(* CODESYS project stepworker_1044.library
   Author: Boido
   Placeholder: StepWorkerLib
   Title: StepWorkerLib
   Version: 1.0.4.4
   Company: FactoryAutomation

Project tree, tasks and I/O mapping:
  libraries: Tc2_Standard, * (Beckhoff Automation GmbH); Tc2_System, * (Beckhoff Automation GmbH); Tc2_Utilities, * (Beckhoff Automation GmbH); Tc3_Module, * (Beckhoff Automation GmbH); VersionLib, * (FactoryAutomation)
  DUTs/
  GVLs/
  POUs/
    function block Actuator [ST]
    function block Boolean [ST]: getValue, setValue
    function block BoolIn [ST]: CallAfterInit, getValue, setValue
    function block BoolOut [ST]: CallAfterInit, getValue, setValue
    function block FB_StepWorker [ST]: getStep, mAddCondition, mConfigureTimeout, mNextStep
    interface I_Comparator: mEquals, mGreaterEquals, mGreaterThan, mLessEquals, mLessThan
    interface I_StepCondition: getValue, setValue
    interface I_StepWorker: mAddCondition
    function block IntComparator [ST]: getValue, mEquals, mGreaterEquals, mGreaterThan, mLessEquals, mLessThan, setValue
    function block LrealComparator [ST]: getValue, mEquals, mGreaterEquals, mGreaterThan, mLessEquals, mLessThan, setValue
    program MAIN [ST]
    function block RealComparator [ST]: getValue, mEquals, mGreaterEquals, mGreaterThan, mLessEquals, mLessThan, setValue
    function block SymbolPathStorage [ST]
    function block UintComparator [ST]: getValue, mEquals, mGreaterEquals, mGreaterThan, mLessEquals, mLessThan, setValue
  VISUs/
  program Version [ST]
*)

// POUs/Actuator
FUNCTION_BLOCK Actuator
VAR_INPUT
END_VAR
VAR_OUTPUT
	fbOutput : BoolOut;
END_VAR
VAR
END_VAR

END_FUNCTION_BLOCK

// POUs/BoolOut
{attribute 'call_after_init'}
{attribute 'reflection'}
FUNCTION_BLOCK PUBLIC BoolOut EXTENDS SymbolPathStorage IMPLEMENTS I_StepCondition
VAR_INPUT
END_VAR
VAR_OUTPUT
END_VAR
VAR
	{attribute 'instance-path'}  
	{attribute 'no_init'} 
	sPath : STRING;
	bValue AT%Q* : BOOL;
	sInitPath : STRING;

END_VAR

{attribute 'call_after_init'}
METHOD PRIVATE CallAfterInit : BOOL
IF uiPathCounter <= cMaxPaths 
THEN
	//Delete the part of the path which contains solution and project name 	
	sInitPath := DELETE(sPath,FIND(sPath,'.'),1);
	sInitPath := DELETE(sInitPath,FIND(sInitPath,'.'),1);
	sInitPath := CONCAT(sInitPath,'.bValue');
	aPaths[uiPathCounter] := sInitPath;
	uiPathCounter := uiPathCounter + 1;
END_IF
END_METHOD


PROPERTY getValue : BOOL
GET
getValue := bValue;
END_GET
END_PROPERTY


PROPERTY setValue : BOOL
SET
bValue := setValue;
END_SET
END_PROPERTY

END_FUNCTION_BLOCK

// POUs/SymbolPathStorage
FUNCTION_BLOCK SymbolPathStorage

VAR_OUTPUT
END_VAR
VAR_STAT
	aPaths : ARRAY[1..cMaxPaths] OF STRING;
	uiPathCounter : UINT := 1;
END_VAR
VAR CONSTANT
	cMaxPaths : UINT := 512;
END_VAR

END_FUNCTION_BLOCK

// POUs/I_StepCondition
INTERFACE I_StepCondition

PROPERTY getValue : BOOL
GET
END_GET
END_PROPERTY

PROPERTY setValue : Bool
SET
END_SET
END_PROPERTY

END_INTERFACE

// POUs/Boolean
FUNCTION_BLOCK PUBLIC Boolean IMPLEMENTS I_StepCondition
VAR_INPUT
END_VAR
VAR_OUTPUT
END_VAR
VAR
	bValue : BOOL;
END_VAR

PROPERTY getValue : BOOL
GET
getValue := bValue;
END_GET
END_PROPERTY


PROPERTY setValue : BOOL
SET
bValue := setValue;
END_SET
END_PROPERTY

END_FUNCTION_BLOCK

// POUs/BoolIn
{attribute 'call_after_init'}
{attribute 'reflection'}
FUNCTION_BLOCK PUBLIC BoolIn EXTENDS SymbolPathStorage IMPLEMENTS I_StepCondition
VAR_INPUT
END_VAR
VAR_OUTPUT
END_VAR
VAR
	
	{attribute 'instance-path'} 
	{attribute 'no_init'} 
	sPath : STRING;
	bValue AT%I* : BOOL;
	sInitPath : STRING;
END_VAR

{attribute 'call_after_init'}
METHOD PRIVATE CallAfterInit : BOOL
IF uiPathCounter <= cMaxPaths 
THEN
	//Delete the part of the path which contains solution and project name 	
	sInitPath := DELETE(sPath,FIND(sPath,'.'),1);
	sInitPath := DELETE(sInitPath,FIND(sInitPath,'.'),1);
	sInitPath := CONCAT(sInitPath,'.bValue');
	aPaths[uiPathCounter] := sInitPath;
	uiPathCounter := uiPathCounter + 1;
END_IF
END_METHOD

{warning 'Eigenschaftenimplementierung hinzufügen'}
PROPERTY getValue : BOOL
GET
getValue := bValue;
END_GET
END_PROPERTY

{warning 'Eigenschaftenimplementierung hinzufügen'}
PROPERTY setValue : BOOL
SET
bValue := setValue;
END_SET
END_PROPERTY

END_FUNCTION_BLOCK

// POUs/FB_StepWorker
FUNCTION_BLOCK PUBLIC FB_StepWorker IMPLEMENTS I_StepWorker
VAR_INPUT
	bResetTimeout : BOOL;
END_VAR
VAR_OUTPUT
	uiStep : UINT;
	bTimeout : BOOL;
END_VAR
VAR
	uiConditionCounter : UINT := 1;
	aConditions	: ARRAY[1..cMaxConditions] OF I_StepCondition;

	bTimeoutFlag : BOOL;	
	fbTimeout : TON;
	tTimeIntern : TIME;
END_VAR
VAR CONSTANT
	cMaxConditions : UINT := 25;
	
END_VAR

IF bResetTimeout
THEN
	bResetTimeout := FALSE;
	bTimeout := FALSE;
	bTimeoutFlag := FALSE;
END_IF

fbTimeout(IN:=bTimeoutFlag, PT:=tTimeIntern , Q=>bTimeout);

PROPERTY getStep : uint
GET
getStep := uiStep;
END_GET
END_PROPERTY

METHOD PUBLIC mAddCondition : I_StepWorker
VAR_INPUT
	itfStepCondition : I_StepCondition;
END_VAR
VAR
	i : UINT;
END_VAR
mAddCondition := THIS^;
IF itfStepCondition = 0
THEN
	//Avoid null pointer exception.
	RETURN;
END_IF

FOR i := 1 TO cMaxConditions DO
	IF aConditions[i] = itfStepCondition 
	THEN
		//Condition already added.
		RETURN;
	END_IF
END_FOR
 
//Add new condition.
aConditions[uiConditionCounter] := itfStepCondition;
uiConditionCounter := uiConditionCounter + 1;
END_METHOD

METHOD mConfigureTimeout : I_StepWorker
VAR_INPUT
	tTime : TIME;
END_VAR
mConfigureTimeout := THIS^;
tTimeIntern := tTime;
bTimeoutFlag := TRUE;
END_METHOD

METHOD mNextStep : UINT
VAR_INPUT
	uiNextStep : UINT;
END_VAR
VAR
	i : UINT;
END_VAR
IF bTimeout
THEN
	mNextStep := uiStep;
	RETURN;
END_IF
	
FOR i := 1 TO (uiConditionCounter-1) DO
	IF aConditions[i].getValue = FALSE 
	THEN
		//1 Condition is false therefor exit.
		mNextStep := uiStep;
		RETURN;
	END_IF
	
END_FOR

//All conditions met
bTimeoutFlag := FALSE;

//Reset the condition counter and conditions
FOR i := 1 TO (uiConditionCounter-1) DO
	aConditions[i] := 0;
END_FOR

uiConditionCounter := 1;
uiStep := uiNextStep;
mNextStep := uiNextStep;
END_METHOD

END_FUNCTION_BLOCK

// POUs/I_StepWorker
INTERFACE I_StepWorker

METHOD PUBLIC mAddCondition : I_StepWorker
VAR_INPUT
	itfStepCondition : I_StepCondition;
END_VAR
END_METHOD

END_INTERFACE

// POUs/I_Comparator
INTERFACE I_Comparator

METHOD mEquals : BOOL;
VAR_INPUT
	rTarget1 : REFERENCE TO UINT;
	rTarget2 : REFERENCE TO UINT;
END_VAR
END_METHOD

METHOD PUBLIC mGreaterEquals : BOOL
VAR_INPUT
	rTarget1 : REFERENCE TO UINT;
	rTarget2 : REFERENCE TO UINT;
END_VAR
END_METHOD

METHOD mGreaterThan : BOOL;
VAR_INPUT
	rTarget1 : REFERENCE TO UINT;
	rTarget2 : REFERENCE TO UINT;
END_VAR
END_METHOD

METHOD mLessEquals : BOOL
VAR_INPUT
	rTarget1 : REFERENCE TO UINT;
	rTarget2 : REFERENCE TO UINT;
END_VAR
END_METHOD

METHOD mLessThan : BOOL;
VAR_INPUT
	rTarget1 : REFERENCE TO UINT;
	rTarget2 : REFERENCE TO UINT;
END_VAR
END_METHOD

END_INTERFACE

// POUs/IntComparator
FUNCTION_BLOCK IntComparator IMPLEMENTS I_Comparator,I_StepCondition
VAR_INPUT
END_VAR
VAR_OUTPUT
END_VAR
VAR
	uiSelector 		: UINT;
	rInternTarget1 	: REFERENCE TO INT;
	rInternTarget2 	: REFERENCE TO INT;
	bValue			: BOOL;
END_VAR

IF NOT __ISVALIDREF( rInternTarget1 )
OR NOT __ISVALIDREF( rInternTarget1 )
THEN
	uiSelector := 0;
END_IF 

CASE uiSelector OF

	0:;
		
	10:
		bValue := mEquals(rInternTarget1,rInternTarget2);
		
	20:
		bValue := mGreaterThan(rInternTarget1,rInternTarget2);
	
	30:
		bValue := mLessThan(rInternTarget1,rInternTarget2);
	
	40:
		bValue := mGreaterEquals(rInternTarget1,rInternTarget2);
		
	50:
		bValue := mLessEquals(rInternTarget1,rInternTarget2);
		
END_CASE

{warning 'Eigenschaftenimplementierung hinzufügen'}
PROPERTY getValue : BOOL
GET
getValue := bValue;
END_GET
END_PROPERTY

METHOD mEquals : BOOL;
VAR_INPUT
	rTarget1 : REFERENCE TO INT;
	rTarget2 : REFERENCE TO INT;
END_VAR
uiSelector := 10;
rInternTarget1 REF= rTarget1;
rInternTarget2 REF= rTarget2;

mEquals := ( rTarget1 = rTarget2 );
END_METHOD

METHOD PUBLIC mGreaterEquals : BOOL
VAR_INPUT
	rTarget1 : REFERENCE TO INT;
	rTarget2 : REFERENCE TO INT;
END_VAR
uiSelector := 40;
rInternTarget1 REF= rTarget1;
rInternTarget2 REF= rTarget2;

mGreaterEquals := ( rTarget1 >= rTarget2 );
END_METHOD

METHOD mGreaterThan : BOOL;
VAR_INPUT
	rTarget1 : REFERENCE TO INT;
	rTarget2 : REFERENCE TO INT;
END_VAR
uiSelector := 20;
rInternTarget1 REF= rTarget1;
rInternTarget2 REF= rTarget2;

mGreaterThan := ( rTarget1 >= rTarget2 );
END_METHOD

METHOD mLessEquals : BOOL
VAR_INPUT
	rTarget1 : REFERENCE TO INT;
	rTarget2 : REFERENCE TO INT;
END_VAR
uiSelector := 50;
rInternTarget1 REF= rTarget1;
rInternTarget2 REF= rTarget2;

mLessEquals := ( rTarget1 <= rTarget2 );
END_METHOD

METHOD mLessThan : BOOL;
VAR_INPUT
	rTarget1 : REFERENCE TO INT;
	rTarget2 : REFERENCE TO INT;
END_VAR
uiSelector := 30;
rInternTarget1 REF= rTarget1;
rInternTarget2 REF= rTarget2;

mLessThan := ( rTarget1 < rTarget2 );
END_METHOD

{warning 'Eigenschaftenimplementierung hinzufügen'}
PROPERTY setValue : BOOL
SET
bValue := setValue;
END_SET
END_PROPERTY

END_FUNCTION_BLOCK

// POUs/LrealComparator
FUNCTION_BLOCK LrealComparator IMPLEMENTS I_Comparator,I_StepCondition
VAR_INPUT
END_VAR
VAR_OUTPUT
END_VAR
VAR
	uiSelector 		: UINT;
	rInternTarget1 	: REFERENCE TO LREAL;
	rInternTarget2 	: REFERENCE TO LREAL;
	bValue			: BOOL;
END_VAR

IF NOT __ISVALIDREF( rInternTarget1 )
OR NOT __ISVALIDREF( rInternTarget1 )
THEN
	uiSelector := 0;
END_IF 

CASE uiSelector OF

	0:;
		
	10:
		bValue := mEquals(rInternTarget1,rInternTarget2);
		
	20:
		bValue := mGreaterThan(rInternTarget1,rInternTarget2);
	
	30:
		bValue := mLessThan(rInternTarget1,rInternTarget2);
	
	40:
		bValue := mGreaterEquals(rInternTarget1,rInternTarget2);
		
	50:
		bValue := mLessEquals(rInternTarget1,rInternTarget2);
		
END_CASE

{warning 'Eigenschaftenimplementierung hinzufügen'}
PROPERTY getValue : BOOL
GET
getValue := bValue;
END_GET
END_PROPERTY

METHOD mEquals : BOOL;
VAR_INPUT
	rTarget1 : REFERENCE TO LREAL;
	rTarget2 : REFERENCE TO LREAL;
END_VAR
uiSelector := 10;
rInternTarget1 REF= rTarget1;
rInternTarget2 REF= rTarget2;

mEquals := ( rTarget1 = rTarget2 );
END_METHOD

METHOD PUBLIC mGreaterEquals : BOOL
VAR_INPUT
	rTarget1 : REFERENCE TO LREAL;
	rTarget2 : REFERENCE TO LREAL;
END_VAR
uiSelector := 40;
rInternTarget1 REF= rTarget1;
rInternTarget2 REF= rTarget2;

mGreaterEquals := ( rTarget1 >= rTarget2 );
END_METHOD

METHOD mGreaterThan : BOOL;
VAR_INPUT
	rTarget1 : REFERENCE TO LREAL;
	rTarget2 : REFERENCE TO LREAL;
END_VAR
uiSelector := 20;
rInternTarget1 REF= rTarget1;
rInternTarget2 REF= rTarget2;

mGreaterThan := ( rTarget1 >= rTarget2 );
END_METHOD

METHOD mLessEquals : BOOL
VAR_INPUT
	rTarget1 : REFERENCE TO LREAL;
	rTarget2 : REFERENCE TO LREAL;
END_VAR
uiSelector := 50;
rInternTarget1 REF= rTarget1;
rInternTarget2 REF= rTarget2;

mLessEquals := ( rTarget1 <= rTarget2 );
END_METHOD

METHOD mLessThan : BOOL;
VAR_INPUT
	rTarget1 : REFERENCE TO LREAL;
	rTarget2 : REFERENCE TO LREAL;
END_VAR
uiSelector := 30;
rInternTarget1 REF= rTarget1;
rInternTarget2 REF= rTarget2;

mLessThan := ( rTarget1 < rTarget2 );
END_METHOD

{warning 'Eigenschaftenimplementierung hinzufügen'}
PROPERTY setValue : BOOL
SET
bValue := setValue;
END_SET
END_PROPERTY

END_FUNCTION_BLOCK

// POUs/MAIN
PROGRAM MAIN
VAR
	fbStepWorker : FB_StepWorker;
	Valve1 : Actuator;
	Valve2 : Actuator;
	Valve3 : Actuator;
	fbUintComparator : UintComparator;
	uiCounter : UINT;
	uiDesiredStep : UINT := 10;
	fbRelease : Boolean;
	bReportTimeout : BOOL;
	test : BOOLIN;
	test2 : BOOLIN;
	sAppName : STRING;
	sProjectName : STRING;
	SystemInfo : PlcAppSystemInfo;
	SymbolPathStorage : SymbolPathStorage;
END_VAR

SystemInfo := _AppInfo;
sAppName := _AppInfo.AppName;
sProjectName := _AppInfo.ProjectName; 

fbUintComparator();
fbStepWorker();

CASE fbStepWorker.uiStep OF

	0:	
	
		fbUintComparator.mEquals(fbStepWorker.uiStep,uiDesiredStep);
		
		fbStepWorker
			.mAddCondition(Valve1.fbOutput)
			.mAddCondition(Valve2.fbOutput)
			.mAddCondition(Valve3.fbOutput);
			
		fbStepWorker.mNextStep(10);
		
		
	10:	
	
		fbStepWorker
			.mConfigureTimeout(T#10S)
			.mAddCondition(fbUintComparator)
			.mAddCondition(fbRelease);
			
		fbStepWorker.mNextStep(20);
		bReportTimeout := fbStepWorker.bTimeout;
		
	20:
		;
	
END_CASE;

END_PROGRAM

// POUs/UintComparator
FUNCTION_BLOCK UintComparator IMPLEMENTS I_Comparator,I_StepCondition
VAR_INPUT
END_VAR
VAR_OUTPUT
END_VAR
VAR
	uiSelector 		: UINT;
	rInternTarget1 	: REFERENCE TO UINT;
	rInternTarget2 	: REFERENCE TO UINT;
	bValue			: BOOL;
END_VAR

IF NOT __ISVALIDREF( rInternTarget1 )
OR NOT __ISVALIDREF( rInternTarget1 )
THEN
	uiSelector := 0;
END_IF 

CASE uiSelector OF

	0:;
		
	10:
		bValue := mEquals(rInternTarget1,rInternTarget2);
		
	20:
		bValue := mGreaterThan(rInternTarget1,rInternTarget2);
	
	30:
		bValue := mLessThan(rInternTarget1,rInternTarget2);
	
	40:
		bValue := mGreaterEquals(rInternTarget1,rInternTarget2);
		
	50:
		bValue := mLessEquals(rInternTarget1,rInternTarget2);
		
END_CASE


PROPERTY getValue : BOOL
GET
getValue := bValue;
END_GET
END_PROPERTY

METHOD mEquals : BOOL;
VAR_INPUT
	rTarget1 : REFERENCE TO UINT;
	rTarget2 : REFERENCE TO UINT;
END_VAR
uiSelector := 10;
rInternTarget1 REF= rTarget1;
rInternTarget2 REF= rTarget2;

mEquals := ( rTarget1 = rTarget2 );
END_METHOD

METHOD PUBLIC mGreaterEquals : BOOL
VAR_INPUT
	rTarget1 : REFERENCE TO UINT;
	rTarget2 : REFERENCE TO UINT;
END_VAR
uiSelector := 40;
rInternTarget1 REF= rTarget1;
rInternTarget2 REF= rTarget2;

mGreaterEquals := ( rTarget1 >= rTarget2 );
END_METHOD

METHOD mGreaterThan : BOOL;
VAR_INPUT
	rTarget1 : REFERENCE TO UINT;
	rTarget2 : REFERENCE TO UINT;
END_VAR
uiSelector := 20;
rInternTarget1 REF= rTarget1;
rInternTarget2 REF= rTarget2;

mGreaterThan := ( rTarget1 >= rTarget2 );
END_METHOD

METHOD mLessEquals : BOOL
VAR_INPUT
	rTarget1 : REFERENCE TO UINT;
	rTarget2 : REFERENCE TO UINT;
END_VAR
uiSelector := 50;
rInternTarget1 REF= rTarget1;
rInternTarget2 REF= rTarget2;

mLessEquals := ( rTarget1 <= rTarget2 );
END_METHOD

METHOD mLessThan : BOOL;
VAR_INPUT
	rTarget1 : REFERENCE TO UINT;
	rTarget2 : REFERENCE TO UINT;
END_VAR
uiSelector := 30;
rInternTarget1 REF= rTarget1;
rInternTarget2 REF= rTarget2;

mLessThan := ( rTarget1 < rTarget2 );
END_METHOD


PROPERTY setValue : BOOL
SET
bValue := setValue;
END_SET
END_PROPERTY

END_FUNCTION_BLOCK

// POUs/RealComparator
FUNCTION_BLOCK RealComparator IMPLEMENTS I_Comparator,I_StepCondition
VAR_INPUT
END_VAR
VAR_OUTPUT
END_VAR
VAR
	uiSelector 		: UINT;
	rInternTarget1 	: REFERENCE TO REAL;
	rInternTarget2 	: REFERENCE TO REAL;
	bValue			: BOOL;
END_VAR

IF NOT __ISVALIDREF( rInternTarget1 )
OR NOT __ISVALIDREF( rInternTarget1 )
THEN
	uiSelector := 0;
END_IF 

CASE uiSelector OF

	0:;
		
	10:
		bValue := mEquals(rInternTarget1,rInternTarget2);
		
	20:
		bValue := mGreaterThan(rInternTarget1,rInternTarget2);
	
	30:
		bValue := mLessThan(rInternTarget1,rInternTarget2);
	
	40:
		bValue := mGreaterEquals(rInternTarget1,rInternTarget2);
		
	50:
		bValue := mLessEquals(rInternTarget1,rInternTarget2);
		
END_CASE

{warning 'Eigenschaftenimplementierung hinzufügen'}
PROPERTY getValue : BOOL
GET
getValue := bValue;
END_GET
END_PROPERTY

METHOD mEquals : BOOL;
VAR_INPUT
	rTarget1 : REFERENCE TO REAL;
	rTarget2 : REFERENCE TO REAL;
END_VAR
uiSelector := 10;
rInternTarget1 REF= rTarget1;
rInternTarget2 REF= rTarget2;

mEquals := ( rTarget1 = rTarget2 );
END_METHOD

METHOD PUBLIC mGreaterEquals : BOOL
VAR_INPUT
	rTarget1 : REFERENCE TO REAL;
	rTarget2 : REFERENCE TO REAL;
END_VAR
uiSelector := 40;
rInternTarget1 REF= rTarget1;
rInternTarget2 REF= rTarget2;

mGreaterEquals := ( rTarget1 >= rTarget2 );
END_METHOD

METHOD mGreaterThan : BOOL;
VAR_INPUT
	rTarget1 : REFERENCE TO REAL;
	rTarget2 : REFERENCE TO REAL;
END_VAR
uiSelector := 20;
rInternTarget1 REF= rTarget1;
rInternTarget2 REF= rTarget2;

mGreaterThan := ( rTarget1 >= rTarget2 );
END_METHOD

METHOD mLessEquals : BOOL
VAR_INPUT
	rTarget1 : REFERENCE TO REAL;
	rTarget2 : REFERENCE TO REAL;
END_VAR
uiSelector := 50;
rInternTarget1 REF= rTarget1;
rInternTarget2 REF= rTarget2;

mLessEquals := ( rTarget1 <= rTarget2 );
END_METHOD

METHOD mLessThan : BOOL;
VAR_INPUT
	rTarget1 : REFERENCE TO REAL;
	rTarget2 : REFERENCE TO REAL;
END_VAR
uiSelector := 30;
rInternTarget1 REF= rTarget1;
rInternTarget2 REF= rTarget2;

mLessThan := ( rTarget1 < rTarget2 );
END_METHOD

{warning 'Eigenschaftenimplementierung hinzufügen'}
PROPERTY setValue : BOOL
SET
bValue := setValue;
END_SET
END_PROPERTY

END_FUNCTION_BLOCK

// Version
PROGRAM Version
VAR
END_VAR

(*

1.0.2.2:	Boido	010120

Added VersionLib and Verstion.txt to the project.

1.0.3.3:	Boido	010120

SymbolPathStorage added to the project.
IO FBs like BoolIn and BoolOut extend SymbolPathStorage in order to have and 
easy way to group all symbol paths in a central storage and make it accessible 
to an ADS interface.

1.0.4.4:	Boido	020120

Version.txt replaced with Version PRG

*)

END_PROGRAM
